FUNCTION_BLOCK TimeOut
VAR_INPUT
	TOutTime : TIME;
END_VAR
VAR
	TIM : Ton;
	Inp : BOOL;
END_VAR

Inp := FALSE;
TIM(IN:=Inp, PT:=TOutTime);

METHOD RunOut : BOOL
VAR_INPUT
	bInp : BOOL;
//	TOutTime : TIME;
END_VAR
Inp :=bInp;
TIM(IN:=Inp, PT:=TOutTime);
RunOut := Tim.Q;
END_METHOD

END_FUNCTION_BLOCK

(* stored: Version 1.1.0.1, ProductVersion 3.1.4024.12
   POU TimeOut: Id {d3d885bb-9bdd-4b88-973a-7c1f9f8608f3}, SpecialFunc None
   Method RunOut: Id {92a3bdde-9d41-4426-826c-37e703a60d27} *)
